// TIA Portal V20 export
VAR_GLOBAL   // PLC tag table "Default tag table"
   Start AT %I0.0 : Bool;
   Stop AT %I0.1 : Bool;
   Program_On AT %Q0.1 : Bool;
   AutoON AT %M100.0 : Bool;   // AutoON
END_VAR
